FUNCTION_BLOCK FB_HE_SATT_FilterCombinationCollector IMPLEMENTS I_HE_SATT_FilterCombinationCollector
VAR CONSTANT
    nMAXIMUM_NUMBER_OF_COMBINATIONS : DINT := 1000;
END_VAR
VAR
    nNumberOfCombinations : DINT;
    afbFilterCombination : ARRAY[1..nMAXIMUM_NUMBER_OF_COMBINATIONS] OF FB_HE_SATT_FilterCombination;
END_VAR


METHOD PUBLIC AddFilterCombination
VAR_INPUT
    fbFilterCombination : REFERENCE TO FB_HE_SATT_FilterCombination;
END_VAR

IF nNumberOfCombinations >= nMAXIMUM_NUMBER_OF_COMBINATIONS THEN
    RETURN;
END_IF

nNumberOfCombinations := nNumberOfCombinations + 1;
afbFilterCombination[nNumberOfCombinations] := fbFilterCombination;
END_METHOD


METHOD GetCombination : REFERENCE TO FB_HE_SATT_FilterCombination
VAR_INPUT
	nCombinationNumber	: DINT;
END_VAR

GetCombination REF= afbFilterCombination[nCombinationNumber];
END_METHOD


PROPERTY NumCombinationsAdded : DINT
GET

NumCombinationsAdded := THIS^.nNumberOfCombinations;
END_GET
END_PROPERTY


METHOD PUBLIC Reset

nNumberOfCombinations := 0;
END_METHOD

END_FUNCTION_BLOCK

(* stored: Version 1.1.0.1
   POU FB_HE_SATT_FilterCombinationCollector: Id {4b240f92-978e-4d19-be0a-9ddef7b6361c}, SpecialFunc None
   Method AddFilterCombination: Id {f4eb5908-4a36-48dd-84ff-a98c52084b57}
   Method GetCombination: Id {faf7cc6b-d99e-4611-9630-58003c4f0463}
   Property NumCombinationsAdded: Id {ad157a5f-587e-40b1-a6f3-2671ffb46be8}
   Get Get: Id {d44944df-ff85-4924-a4fe-41bc08897ab9}
   Method Reset: Id {912b6c75-b835-4fa2-8b93-0deeceaaf550} *)
